TYPE ST_peakshavebox_params :
STRUCT
	PSBhardware			: ePSBhardware := ePSBHardware.Beckhoff; // if enabled, psb v2 is configured.
	fastmode 			: BOOL := TRUE; // only in old PSB
END_STRUCT
END_TYPE

(* stored: Version 1.1.0.1, ProductVersion 3.1.4024.12
   DUT ST_peakshavebox_params: Id {905fe61c-a96c-43f5-9976-24ad1ecff638} *)
